PROGRAM POS_Comparition
VAR
	fbPOS_ComparitionXY:FB_013_POS_Comparition;
	fbPOS_ComparitionZR:FB_013_POS_Comparition;
END_VAR

// XY位置比较
fbPOS_ComparitionXY(arstCamCtrl:=arstCamCtrlIO, fbstIJP:=stIJP , stAxis:=arstAxis );

END_PROGRAM

(* stored: Version 1.1.0.1, ProductVersion 3.1.4024.12
   POU POS_Comparition: Id {d9ece25e-1ad1-47ae-9f0c-1b04546361ef}, SpecialFunc None *)
